TYPE ST_Counter :
STRUCT
	//Counter Overall/Shift
	diOverallCounterOk	: UDINT;
	diOverallCounterNok	: UDINT;
END_STRUCT
END_TYPE

(* stored: Version 1.1.0.1, ProductVersion 3.1.4024.11
   DUT ST_Counter: Id {da56201e-bd28-4dac-8de7-be99aee690d1} *)
